TYPE ST_ReceiveTestStatus :
STRUCT
	TransmitDone        :BOOL;   //数据发送完成
    ReceiveRequest      :BOOL;    
    InitAccepted        :BOOL;
    SndBufferFull       :BOOL;
    PutDataDone         :BOOL;
    InputLength         :USINT;
    TotalInputLength    :UINT;
END_STRUCT
END_TYPE

(* stored: Version 1.1.0.1, ProductVersion 3.1.4024.9
   DUT ST_ReceiveTestStatus: Id {cfd31f5c-6029-448d-b20e-b191953f3ed0} *)
